(* PLC project Untitled1, Beckhoff Automation GmbH TF6420 Database Server Query Analyser 1.0.0.0 *)
(* stored: creationDateTime 2018-10-18T13:42:14, modificationDateTime 2018-10-18T13:42:14 *)

TYPE ST_SelectStruct : STRUCT
  time : LINT;
  Temperature : LREAL;
  ID : LINT;
  name : STRING(255);
  humidity : LREAL;
  CO2 : LREAL;
  Light1 : INT;
  Light2 : INT;
  Light3 : INT;
  Light4 : INT;
  AnalogAux1 : LINT;
  AnalogAux2 : LINT;
  AnalogAux3 : LINT;
  AnalogAux4 : LINT;
  DigitalAux1 : BOOL;
  DigitalAux2 : BOOL;
  DigitalAux3 : BOOL;
  DigitalAux4 : BOOL;
END_STRUCT;
END_TYPE
